// TIA Portal project "ChemicalProcess" (V16)

(* hardware
DEVICE "S71500/ET200MP station_1"  S7-1500 station
   slot 0: "Rail_0"  Rack  6ES7 590-1***0-0AA0
   slot 0: "PS 25W 24VDC_1"  PS 25W 24VDC  6ES7 505-0KA00-0AB0  V1.0
   slot 1: "PLC_1"  CPU 1511-1 PN  6ES7 511-1AK01-0AB0  V2.8
      slot 3: "CPU display_1"  6ES7591-1AA00-0AA0
      slot 32768: "PROFINET interface_1"  X1
         slot 32769: "Port_1"  X1 P1
         slot 32770: "Port_2"  X1 P2
      slot 34817: "Virtual CP interface port_1"  Virtual CP interface port  Virtual CP interface port
   slot 2: "DI 16x24VDC BA_1"  DI 16x24VDC BA  6ES7 521-1BH10-0AA0  V1.1
   slot 3: "DQ 16x24VDC/0.5A BA_1"  DQ 16x24VDC/0.5A BA  6ES7 522-1BH10-0AA0  V1.1
   slot 4: "AI 8xU/I/RTD/TC ST_1"  AI 8xU/I/RTD/TC ST  6ES7 531-7KF00-0AB0  V2.2
   slot 5: "AQ 2xU/I ST_1"  AQ 2xU/I ST  6ES7 532-5NB00-0AB0  V1.0
   slot 6: "DI 16x24VDC BA_2"  DI 16x24VDC BA  6ES7 521-1BH10-0AA0  V1.1
DEVICE "HMI_1"  KTP700 Basic PN
   slot 0: "HMI_1"  KTP700 Basic PN  6AV2 123-2GB03-0AX0  16.0.0.0
   slot 1: "HMI_RT_1"  KTP700 Basic PN  6AV2 123-2GB03-0AX0  16.0.0.0
   slot 5: "HMI_1.IE_CP_1"  PROFINET Interface  16.0.0.0
      slot 1: "PROFINET Interface_1"  PROFINET Interface
         slot 1: "Port_1"  Port
*)

// ===== PLC "PLC_1"  CPU 1511-1 PN =====

VAR_GLOBAL   // PLC tag table "Default tag table"
   "Start" AT %I12.0 : Bool;
   "Stop" AT %I12.1 : Bool;
   "FICSetpoint" AT %MD14 : Real;
END_VAR

VAR_GLOBAL   // PLC tag table "SIMIT interface"
   "ZSO-510" AT %I0.0 : Bool;
   "ZSC-510" AT %I0.1 : Bool;
   "ZSO-511" AT %I0.2 : Bool;
   "ZSC-511" AT %I0.3 : Bool;
   "ZSO-514" AT %I0.4 : Bool;
   "ZSC-514" AT %I0.5 : Bool;
   "ZSO-519" AT %I0.6 : Bool;
   "ZSC-519" AT %I0.7 : Bool;
   "ZSO-521" AT %I1.0 : Bool;
   "ZSC-521" AT %I1.1 : Bool;
   "M001.R" AT %I1.2 : Bool;
   "M002.R" AT %I1.3 : Bool;
   "LS-513" AT %I1.4 : Bool;
   "GSV-510" AT %Q0.0 : Bool;
   "GSV-511" AT %Q0.1 : Bool;
   "GSV-514" AT %Q0.2 : Bool;
   "GSV-519" AT %Q0.3 : Bool;
   "GSV-521" AT %Q0.4 : Bool;
   "M001.ST" AT %Q0.5 : Bool;
   "M002.ST" AT %Q0.6 : Bool;
   "WT-512" AT %IW2 : Int;
   "LT-515" AT %IW4 : Int;
   "FT-516" AT %IW6 : Int;
   "TT-517" AT %IW8 : Int;
   "TT-518" AT %IW10 : Int;
   "M003.SP" AT %QW2 : Int;
   "M001.F" AT %I1.5 : Bool;
   "M002.F" AT %I1.6 : Bool;
   "M003.R" AT %I1.7 : Bool;
   "M003.F" AT %I18.0 : Bool;
   "M003.ST" AT %Q0.7 : Bool;
   "M001.TK" AT %I18.1 : Bool;
   "M002.TK" AT %I18.2 : Bool;
   "M003.TK" AT %I18.3 : Bool;
END_VAR

DATA_BLOCK "ProcessSequence_DB"   // DB3
{ S7_Optimized_Access := 'TRUE' }
VERSION : 0.1
// stored: InstanceOfName ProcessSequence
"ProcessSequence"
BEGIN
END_DATA_BLOCK

DATA_BLOCK "DB_TestMode"   // DB24
{ S7_Optimized_Access := 'TRUE' }
VERSION : 0.1
// stored: InstanceOfName FB_TestMode
"FB_TestMode"
BEGIN
END_DATA_BLOCK

// folder: Motors/Data Blocks

DATA_BLOCK "DB_M001"   // DB10
{ S7_Optimized_Access := 'TRUE' }
VERSION : 0.1
// stored: InstanceOfName FB_Motor
"FB_Motor"
BEGIN
END_DATA_BLOCK

DATA_BLOCK "DB_M002"   // DB14
{ S7_Optimized_Access := 'TRUE' }
VERSION : 0.1
// stored: InstanceOfName FB_Motor
"FB_Motor"
BEGIN
END_DATA_BLOCK

DATA_BLOCK "DB_M003"   // DB18
{ S7_Optimized_Access := 'TRUE' }
VERSION : 0.1
// stored: InstanceOfName FB_Motor
"FB_Motor"
BEGIN
END_DATA_BLOCK

// folder: Process/Data Blocks

DATA_BLOCK "DB_HMI"   // DB19
{ S7_Optimized_Access := 'TRUE' }
VERSION : 0.1
// stored: InstanceOfName FB_HMI
"FB_HMI"
BEGIN
END_DATA_BLOCK

DATA_BLOCK "DB_AutoMode"   // DB20
{ S7_Optimized_Access := 'TRUE' }
VERSION : 0.1
// stored: InstanceOfName FB_Auto
"FB_Auto"
BEGIN
END_DATA_BLOCK

DATA_BLOCK "DB_ManualMode"   // DB21
{ S7_Optimized_Access := 'TRUE' }
VERSION : 0.1
// stored: InstanceOfName FB_Manual
"FB_Manual"
BEGIN
END_DATA_BLOCK

DATA_BLOCK "DB_Stop"   // DB22
{ S7_Optimized_Access := 'TRUE' }
VERSION : 0.1
// stored: InstanceOfName FB_EStop
"FB_EStop"
BEGIN
END_DATA_BLOCK

DATA_BLOCK "DB_Fault"   // DB23
{ S7_Optimized_Access := 'TRUE' }
VERSION : 0.1
// stored: InstanceOfName FB_Fault
"FB_Fault"
BEGIN
END_DATA_BLOCK

// folder: Sensors/DataBlocks

DATA_BLOCK "DB_Sensor_FIC_516"   // DB4
{ S7_Optimized_Access := 'TRUE' }
VERSION : 0.1
// stored: InstanceOfName SensorScaling
"SensorScaling"
BEGIN
END_DATA_BLOCK

DATA_BLOCK "DB_Sensor_WI_512"   // DB12
{ S7_Optimized_Access := 'TRUE' }
VERSION : 0.1
// stored: InstanceOfName SensorScaling
"SensorScaling"
BEGIN
END_DATA_BLOCK

DATA_BLOCK "DB_Sensor_LI_515"   // DB15
{ S7_Optimized_Access := 'TRUE' }
VERSION : 0.1
// stored: InstanceOfName SensorScaling
"SensorScaling"
BEGIN
END_DATA_BLOCK

DATA_BLOCK "Db_Sensor_TI_517"   // DB16
{ S7_Optimized_Access := 'TRUE' }
VERSION : 0.1
// stored: InstanceOfName SensorScaling
"SensorScaling"
BEGIN
END_DATA_BLOCK

DATA_BLOCK "DB_Sensor_TI_518"   // DB17
{ S7_Optimized_Access := 'TRUE' }
VERSION : 0.1
// stored: InstanceOfName SensorScaling
"SensorScaling"
BEGIN
END_DATA_BLOCK

// folder: System blocks/Program resources

DATA_BLOCK "MixTankMotorTImer"   // DB2
{ S7_Optimized_Access := 'TRUE' }
AUTHOR : Simatic
FAMILY : IEC
NAME : IEC_TMR
VERSION : 1.0
// stored: InstanceOfName IEC_TIMER
"IEC_TIMER"
BEGIN
END_DATA_BLOCK

// folder: Valves/DataBlock_Valves

DATA_BLOCK "DB_GSV_510"   // DB5
{ S7_Optimized_Access := 'TRUE' }
VERSION : 0.1
// stored: InstanceOfName FB_Valve
"FB_Valve"
BEGIN
END_DATA_BLOCK

DATA_BLOCK "DB_GSV_511"   // DB6
{ S7_Optimized_Access := 'TRUE' }
VERSION : 0.1
// stored: InstanceOfName FB_Valve
"FB_Valve"
BEGIN
END_DATA_BLOCK

DATA_BLOCK "DB_GSV_514"   // DB7
{ S7_Optimized_Access := 'TRUE' }
VERSION : 0.1
// stored: InstanceOfName FB_Valve
"FB_Valve"
BEGIN
END_DATA_BLOCK

DATA_BLOCK "DB_GSV_519"   // DB8
{ S7_Optimized_Access := 'TRUE' }
VERSION : 0.1
// stored: InstanceOfName FB_Valve
"FB_Valve"
BEGIN
END_DATA_BLOCK

DATA_BLOCK "DB_GSV_521"   // DB9
{ S7_Optimized_Access := 'TRUE' }
VERSION : 0.1
// stored: InstanceOfName FB_Valve
"FB_Valve"
BEGIN
END_DATA_BLOCK

// folder: (top level)

FUNCTION_BLOCK "ProcessSequence"   // FB1, GRAPH_PLUS
{ S7_Optimized_Access := 'TRUE' }
VERSION : 0.1
   VAR_INPUT
      WI_512 : Real;   // WT-512 is Weight Sensor and connected in OB
      LSA_513 : Bool;   // LS-513 Powder Low level Button
      SetTimeForMixing : Time;   // MIx Tank Motor timing
      TI_517 : Real;
      TI_518 : Real;
      FIC_516 : Real;   // FIC-516 is Pressure sensor Integrated with M003
      LI_515 : Real;   // LT-515 Level indicative sensor
      ACK_EF : Bool := false;   // Acknowledge all errors and faults
      Auto : Bool;   // Automode makes sytem run automatically until pressed stop.
      Manual : Bool;   // Manual mode make user start everytime time the storage tank is emptied.
      M003_SP : Real;   // PIDTulo
   END_VAR
   VAR_OUTPUT
      Initiate : Bool;   // Start initiates the program
      HS_510_Open : Bool;   // ZSC-510 is Valve open signal GSV-510.
      HS_510_Close : Bool;   // ZSC-510 Valve close signal for GSV-510.
      GSV_510 : Bool;   // GSV_510 Valve
      HS_511_Open_ : Bool;   // ZSO-511 is Valve open signal GSV-511.
      HS_511_Close : Bool;   // ZSC-511 Valve close signal
      GSV_511 : Bool;   // GSV-511 Valve
      HS_514_Open : Bool;   // ZSO-514 is Valve open signal for GSV-514
      HS_514_Close : Bool;   // ZSC-514 is valve close signal for GSV-514
      GSV_514 : Bool;   // Valve GSV-514.
      HS_519_Open : Bool;   // ZSO-519 is valve open signal for GSV-519
      HS_519_Close : Bool;   // ZSC-519 is Valve close signal for GSV-519
      GSV_519 : Bool;
      HS_521_Open : Bool;   // ZSO-521 valve open signal for GSV-521
      HS_521_Close : Bool;   // ZSC-521 close valve signal for GSV_521
      GSV_521 : Bool;
      SetElapseTimeforMixing : Time;   // Elaspse time for mix tank motor
      M001_ST : Bool;   // M001.ST is Powder Motor start signal.
      M001_TK : Bool;   // M001.TK is Temperature protection of POwder Motor.
      M001_F : Bool;   // M001.F fault signal of Powder Motor
      M001_R : Bool;   // Reset of Powder Motor
      M002_ST : Bool;   // M002.ST is Mixtank Motor signal.
      M002_TK : Bool;
      M002_F : Bool;   // Mator Fault signal For Mix Tank motor
      M002_R : Bool;   // Reset for Mixing Motor
      M003_ST : Bool;   // M003.ST is Start signal of Motor M003
      M003_F : Bool;   // M003.F is Fault signal of Motor M003
      M003_TK : Bool;   // M003.TK isTemperature protection signal of Motor M003
      M003_R : Bool;   // M003.R is Reset signal of Motor M003
      StopandWait : Bool;   // Stop the Process and goest back S and wait until pressed start manually
   END_VAR
   VAR
      HMI_INFO : Array[0..22] of UInt;
      IF_PAR : G7_IfParPlus_V6;
      RT_DATA : G7_RTDataPlus_V6;   // Internal data area
      Trans1 : G7_TransitionPlus_V6;   // Transition structure
      Trans2 : G7_TransitionPlus_V6;   // Transition structure
      Trans3 : G7_TransitionPlus_V6;   // Transition structure
      Trans4 : G7_TransitionPlus_V6;   // Transition structure
      Trans5 : G7_TransitionPlus_V6;   // Transition structure
      Trans6 : G7_TransitionPlus_V6;   // Transition structure
      Trans7 : G7_TransitionPlus_V6;   // Transition structure
      Trans8 : G7_TransitionPlus_V6;   // Transition structure
      Trans9 : G7_TransitionPlus_V6;   // Transition structure
      Trans10 : G7_TransitionPlus_V6;   // Transition structure
      Trans11 : G7_TransitionPlus_V6;   // Transition structure
      Trans12 : G7_TransitionPlus_V6;   // Transition structure
      Start : G7_StepPlus_V6;   // Step structure
      "Fill NaOH" : G7_StepPlus_V6;   // Step structure
      "Fill Powder M001" : G7_StepPlus_V6;   // Step structure
      "Start Mixing" : G7_StepPlus_V6;   // Step structure
      "Empty MIX Tank" : G7_StepPlus_V6;   // Step structure
      "Stop Water" : G7_StepPlus_V6;   // Step structure
      "Close NaOH valve" : G7_StepPlus_V6;   // Step structure
      "Powder Motor Stop" : G7_StepPlus_V6;   // Step structure
      "Stop Mixing" : G7_StepPlus_V6;   // Step structure
      "Empty Storage Tank" : G7_StepPlus_V6;   // Step structure
      "Stop emptying" : G7_StepPlus_V6;   // Step structure
      "Exit valve open" : G7_StepPlus_V6;   // Step structure
      Step13 : G7_StepPlus_V6;   // Step structure
      "Not to Storage" : G7_StepPlus_V6;   // Step structure
      "Exit valve close" : G7_StepPlus_V6;   // Step structure
      "Valve 521 Stays open" : G7_StepPlus_V6;   // Step structure
      "Fill water" : G7_StepPlus_V6;   // Step structure
      Step18 : G7_StepPlus_V6;   // Step structure
      SINI : Array[0..15] of USInt;
      LSTT : Array[0..11] of USInt;
      ATAJ : Array[0..11] of USInt;
      ATAB : Array[0..11] of USInt;
      PSTT : Array[0..11] of USInt;
      NSTT : Array[0..11] of USInt;
      ASSJ : Array[0..17] of USInt;
      ASSB : Array[0..17] of USInt;
      PTTS : Array[0..17] of USInt;
      NTTS : Array[0..17] of USInt;
      SW_SQTS : Array[0..17] of USInt;
      SWITCH : Array[0..36] of USInt;
      TVX : Array[0..15] of USInt;
      TTX : Array[0..15] of USInt;
      TSX : Array[0..15] of USInt;
      S00X : Array[0..15] of USInt;
      SOFFX : Array[0..15] of USInt;
      SONX : Array[0..15] of USInt;
      SAX : Array[0..15] of USInt;
      SERRX : Array[0..18] of USInt;
      SMX : Array[0..18] of USInt;
      S0X : Array[0..18] of USInt;
      S1X : Array[0..18] of USInt;
      IL_ALARM_INST : Diag_Alarm;
      SUP_ALARM_INST : Diag_Alarm;
      STEP_TIME_ALARM_INST : Diag_Alarm;
      IEC_TIMER_INST : IEC_TIMER;
      TRANSACTION_FLAG : Bool := false;
   END_VAR
   // SINI[0] := 2;
   // SINI[2] := 255;
   // SINI[3] := 255;
   // SINI[4] := 255;
   // SINI[5] := 255;
   // SINI[6] := 255;
   // SINI[7] := 255;
   // SINI[8] := 255;
   // SINI[9] := 255;
   // SINI[10] := 255;
   // SINI[11] := 255;
   // SINI[12] := 255;
   // SINI[13] := 255;
   // SINI[14] := 255;
   // SINI[15] := 255;
   // LSTT[0] := 255;
   // LSTT[1] := 255;
   // LSTT[2] := 255;
   // LSTT[3] := 255;
   // LSTT[4] := 255;
   // LSTT[5] := 255;
   // LSTT[7] := 255;
   // LSTT[8] := 255;
   // ATAJ[1] := 1;
   // ATAJ[2] := 2;
   // ATAJ[3] := 3;
   // ATAJ[4] := 4;
   // ATAJ[5] := 5;
   // ATAJ[6] := 6;
   // ATAJ[7] := 7;
   // ATAJ[8] := 8;
   // ATAJ[9] := 9;
   // ATAB[1] := 1;
   // ATAB[2] := 2;
   // ATAB[3] := 3;
   // ATAB[4] := 4;
   // ATAB[5] := 5;
   // ATAB[6] := 6;
   // ATAB[7] := 7;
   // ATAB[8] := 8;
   // ATAB[9] := 9;
   // PSTT[1] := 1;
   // PSTT[2] := 2;
   // PSTT[3] := 3;
   // PSTT[4] := 4;
   // PSTT[5] := 9;
   // PSTT[6] := 10;
   // PSTT[7] := 11;
   // PSTT[8] := 12;
   // PSTT[9] := 14;
   // NSTT[0] := 16;
   // NSTT[1] := 2;
   // NSTT[2] := 3;
   // NSTT[3] := 4;
   // NSTT[4] := 9;
   // NSTT[5] := 11;
   // NSTT[7] := 12;
   // NSTT[8] := 14;
   // ASSJ[1] := 5;
   // ASSJ[2] := 6;
   // ASSJ[3] := 7;
   // ASSJ[4] := 8;
   // ASSJ[5] := 1;
   // ASSJ[6] := 2;
   // ASSJ[7] := 3;
   // ASSJ[8] := 4;
   // ASSJ[9] := 9;
   // ASSJ[10] := 10;
   // ASSJ[11] := 13;
   // ASSJ[12] := 12;
   // ASSJ[13] := 11;
   // ASSJ[14] := 15;
   // ASSJ[15] := 14;
   // ASSB[1] := 5;
   // ASSB[2] := 6;
   // ASSB[3] := 7;
   // ASSB[4] := 8;
   // ASSB[5] := 1;
   // ASSB[6] := 2;
   // ASSB[7] := 3;
   // ASSB[8] := 4;
   // ASSB[9] := 10;
   // ASSB[10] := 9;
   // ASSB[11] := 13;
   // ASSB[12] := 12;
   // ASSB[13] := 11;
   // ASSB[14] := 15;
   // ASSB[15] := 14;
   // PTTS[0] := 255;
   // PTTS[2] := 1;
   // PTTS[3] := 2;
   // PTTS[4] := 3;
   // PTTS[6] := 1;
   // PTTS[7] := 2;
   // PTTS[8] := 3;
   // PTTS[9] := 4;
   // PTTS[10] := 4;
   // PTTS[11] := 5;
   // PTTS[12] := 7;
   // PTTS[13] := 5;
   // PTTS[14] := 8;
   // PTTS[15] := 8;
   // NTTS[1] := 1;
   // NTTS[2] := 2;
   // NTTS[3] := 3;
   // NTTS[4] := 4;
   // NTTS[5] := 1;
   // NTTS[6] := 2;
   // NTTS[7] := 3;
   // NTTS[8] := 4;
   // NTTS[9] := 5;
   // NTTS[10] := 6;
   // NTTS[11] := 7;
   // NTTS[12] := 8;
   // NTTS[13] := 7;
   // NTTS[14] := 9;
   // NTTS[15] := 9;
   // SW_SQTS[1] := 1;
   // SW_SQTS[2] := 2;
   // SW_SQTS[3] := 3;
   // SW_SQTS[4] := 4;
   // SW_SQTS[5] := 5;
   // SW_SQTS[6] := 6;
   // SW_SQTS[7] := 7;
   // SW_SQTS[8] := 8;
   // SW_SQTS[9] := 9;
   // SW_SQTS[10] := 10;
   // SW_SQTS[11] := 11;
   // SW_SQTS[12] := 12;
   // SW_SQTS[13] := 13;
   // SW_SQTS[14] := 14;
   // SW_SQTS[15] := 15;
   // SWITCH[2] := 64;
   // SWITCH[5] := 1;
   // SWITCH[7] := 4;
   // SWITCH[9] := 16;
   // SWITCH[10] := 64;
   // SWITCH[13] := 1;
   // SWITCH[15] := 4;
   // SWITCH[17] := 16;
   // SWITCH[20] := 8;
   // SWITCH[22] := 232;
   // SWITCH[23] := 7;
   // SWITCH[25] := 1;
   // SWITCH[28] := 128;
   // SWITCH[29] := 1;
   // SWITCH[31] := 33;
   // TVX[0] := 16#1;
   // TTX[0] := 16#1;
   // TSX[0] := 16#1;
   // S00X[0] := 16#1;
   // SOFFX[0] := 16#1;
   // SONX[0] := 16#1;
   // SAX[0] := 16#1;
   // SERRX[0] := 16#1;
   // SMX[0] := 16#1;
   // S0X[0] := 16#1;
   // S1X[0] := 16#1;
   // LSTT[10] := 255;
   // ATAJ[10] := 10;
   // ATAB[10] := 10;
   // PSTT[10] := 16;
   // NSTT[10] := 1;
   // ASSJ[16] := 16;
   // ASSB[16] := 16;
   // PTTS[1] := 10;
   // PTTS[5] := 10;
   // NTTS[16] := 10;
   // LSTT[9] := 255;
   // ATAJ[11] := 11;
   // ATAB[11] := 11;
   // PSTT[11] := 17;
   // NSTT[9] := 17;
   // ASSJ[17] := 17;
   // ASSB[17] := 17;
   // PTTS[17] := 9;
   // NTTS[17] := 11;
   // SW_SQTS[17] := 16;
   // SWITCH[24] := 32;
   // SWITCH[26] := 64;
   // SWITCH[33] := 34;
   // SWITCH[35] := 4;
BEGIN
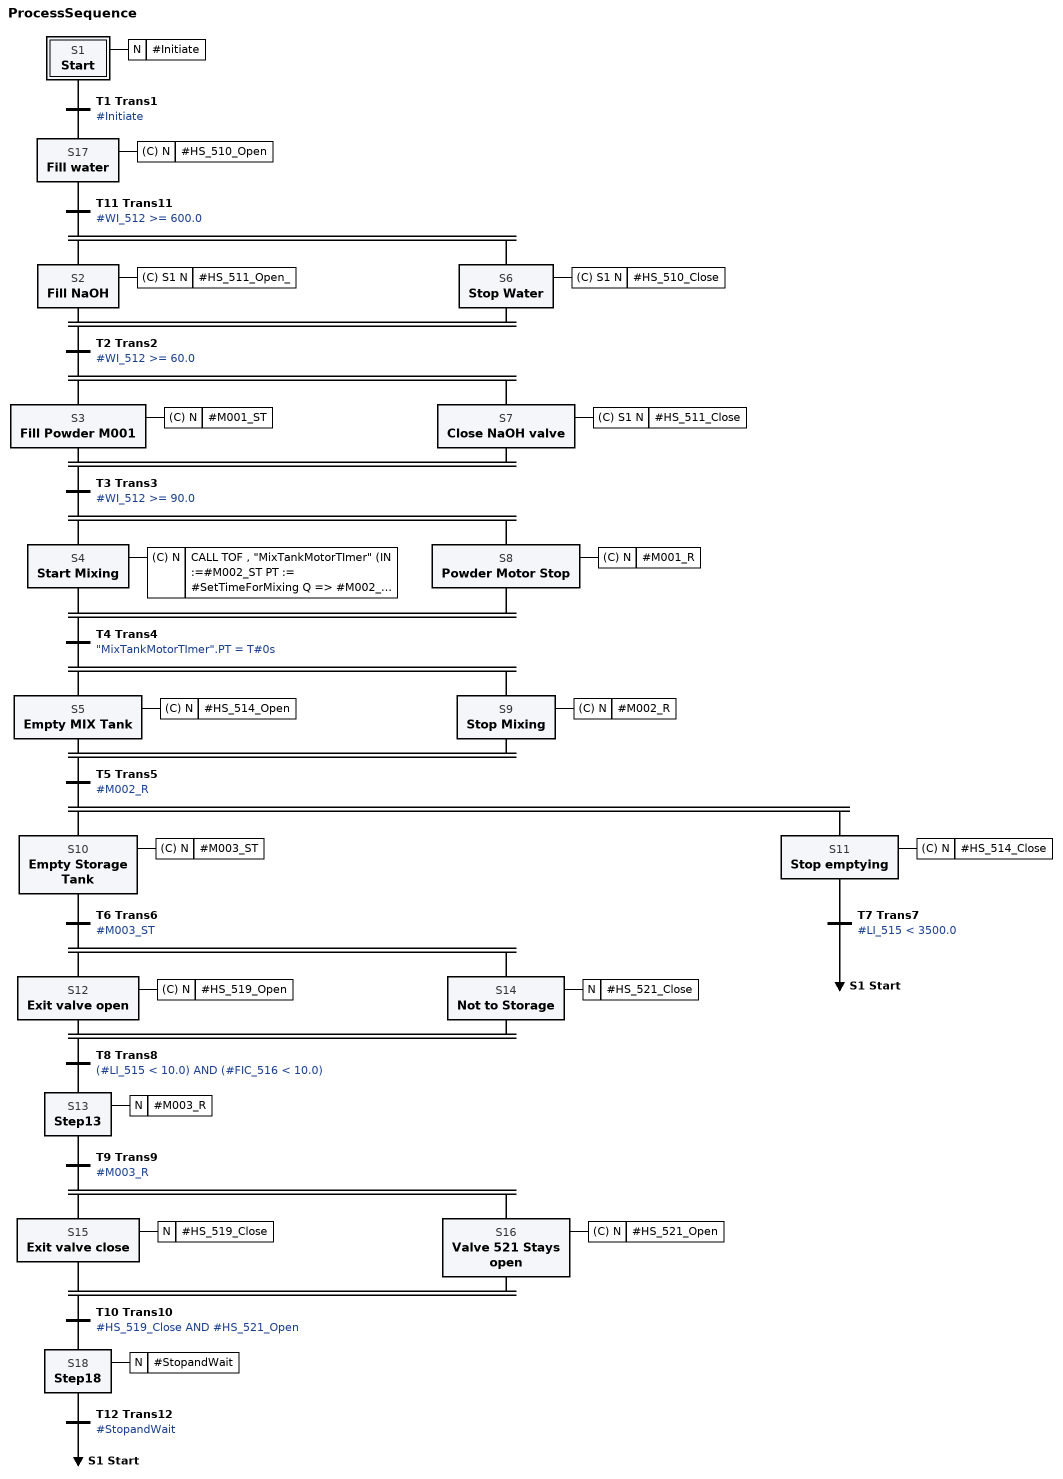
   // sequencer 1
   INITIAL_STEP Start:   // S1, max time T#10S, warning time T#7S
      interlock C := ((#Auto AND NOT #Manual) OR (#Manual AND NOT #Auto)) AND NOT #StopandWait;
              N    #Initiate
   END_STEP
   TRANSITION Trans1 FROM Start TO "Fill water"   // T1
      := #Initiate;
   END_TRANSITION
   STEP "Fill NaOH":   // S2, max time T#10S, warning time T#7S
      interlock C := (#WI_512 <= 40.0) AND NOT #GSV_510 AND NOT #M001_ST AND NOT #M002_ST;
      // 600Kg to 1200kg in weight sensor is 600Kg of NaOH.
      (C) S1  N    #HS_511_Open_
   END_STEP
   STEP "Fill Powder M001":   // S3, max time T#10S, warning time T#7S
      interlock C := NOT #GSV_510 AND NOT #M002_ST AND NOT #LSA_513 AND NOT #M001_F AND NOT #M001_TK AND NOT #GSV_511;
      // 1200-1800KG in wight sensor = 600Kg of Powder
      (C)     N    #M001_ST
   END_STEP
   STEP "Start Mixing":   // S4, max time T#10S, warning time T#7S
      interlock C := NOT #GSV_510 AND NOT #GSV_511 AND NOT #M001_ST AND NOT #M002_F;
      (C)     N    CALL TOF , "MixTankMotorTImer"
                   (IN :=#M002_ST
                   PT := #SetTimeForMixing
                   Q => #M002_R
                   ET=> #SetElapseTimeforMixing
                   )
   END_STEP
   STEP "Empty MIX Tank":   // S5, max time T#10S, warning time T#7S
      interlock C := (#LI_515 < 80.0) AND NOT #GSV_510 AND NOT #GSV_511 AND NOT #M002_ST AND NOT #M001_ST;
      (C)     N    #HS_514_Open
   END_STEP
   STEP "Stop Water":   // S6, max time T#10S, warning time T#7S
      interlock C := #WI_512 >= 30.0;
      // If Valve opens have to make sure it closes.
      (C) S1  N    #HS_510_Close
   END_STEP
   TRANSITION Trans2 FROM ("Fill NaOH", "Stop Water") TO ("Fill Powder M001", "Close NaOH valve")   // T2
      := #WI_512 >= 60.0;
   END_TRANSITION
   STEP "Close NaOH valve":   // S7, max time T#10S, warning time T#7S
      interlock C := #WI_512 = 60.0;
      (C) S1  N    #HS_511_Close
   END_STEP
   TRANSITION Trans3 FROM ("Fill Powder M001", "Close NaOH valve") TO ("Start Mixing", "Powder Motor Stop")   // T3
      := #WI_512 >= 90.0;
   END_TRANSITION
   STEP "Powder Motor Stop":   // S8, max time T#10S, warning time T#7S
      interlock C := #WI_512 >= 90.0;
      (C)     N    #M001_R
   END_STEP
   TRANSITION Trans4 FROM ("Start Mixing", "Powder Motor Stop") TO ("Empty MIX Tank", "Stop Mixing")   // T4
      := "MixTankMotorTImer".PT = T#0s;
   END_TRANSITION
   STEP "Stop Mixing":   // S9, max time T#10S, warning time T#7S
      interlock C := "MixTankMotorTImer".PT = T#0s;
      (C)     N    #M002_R
   END_STEP
   TRANSITION Trans5 FROM ("Empty MIX Tank", "Stop Mixing") TO ("Empty Storage Tank", "Stop emptying")   // T5
      := #M002_R;
   END_TRANSITION
   STEP "Empty Storage Tank":   // S10, max time T#10S, warning time T#7S
      interlock C := NOT #GSV_514 AND (#LI_515 > 70.0) AND NOT #M003_F AND NOT #M003_TK AND NOT #M003_R;
      (C)     N    #M003_ST
   END_STEP
   TRANSITION Trans6 FROM "Empty Storage Tank" TO ("Exit valve open", "Not to Storage")   // T6
      := #M003_ST;
   END_TRANSITION
   STEP "Stop emptying":   // S11, max time T#10S, warning time T#7S
      interlock C := #WI_512 <= 2.0;   // Stop Emptying
      (C)     N    #HS_514_Close
   END_STEP
   TRANSITION Trans7 FROM "Stop emptying" TO Start   // T7, jump
      := #LI_515 < 3500.0;
   END_TRANSITION
   STEP "Exit valve open":   // S12, max time T#10S, warning time T#7S
      interlock C := #M003_ST;
      (C)     N    #HS_519_Open
   END_STEP
   STEP Step13:   // S13, max time T#10S, warning time T#7S
      interlock C := (#LI_515 < 5.0) AND (#FIC_516 < 5.0);
              N    #M003_R
   END_STEP
   TRANSITION Trans9 FROM Step13 TO ("Exit valve close", "Valve 521 Stays open")   // T9
      := #M003_R;
   END_TRANSITION
   STEP "Not to Storage":   // S14, max time T#10S, warning time T#7S
      interlock C := #M003_ST;
              N    #HS_521_Close
   END_STEP
   TRANSITION Trans8 FROM ("Exit valve open", "Not to Storage") TO Step13   // T8
      := (#LI_515 < 10.0) AND (#FIC_516 < 10.0);
   END_TRANSITION
   STEP "Exit valve close":   // S15, max time T#10S, warning time T#7S
      interlock C := #M003_R AND (#FIC_516 < 5.0);
              N    #HS_519_Close
   END_STEP
   STEP "Valve 521 Stays open":   // S16, max time T#10S, warning time T#7S
      interlock C := #M003_R AND (#FIC_516 < 5.0);
      (C)     N    #HS_521_Open
   END_STEP
   TRANSITION Trans10 FROM ("Exit valve close", "Valve 521 Stays open") TO Step18   // T10
      := #HS_519_Close AND #HS_521_Open;
   END_TRANSITION
   STEP "Fill water":   // S17, max time T#10S, warning time T#7S
      interlock C := (#WI_512 <= 5.0) AND NOT #HS_510_Close AND NOT #GSV_511 AND NOT #M001_ST AND NOT #M002_ST;
      // 1Litre = 1Kg, 0-600Kg in Weight sensor is 600litres of Water For forcing value of sensors converts kg value to Siemens analog raw value (0...27648). For 200KG = 2765
      (C)     N    #HS_510_Open
   END_STEP
   TRANSITION Trans11 FROM "Fill water" TO ("Fill NaOH", "Stop Water")   // T11
      := #WI_512 >= 600.0;
   END_TRANSITION
   STEP Step18:   // S18, max time T#10S, warning time T#7S
              N    #StopandWait
   END_STEP
   TRANSITION Trans12 FROM Step18 TO Start   // T12, jump
      := #StopandWait;
   END_TRANSITION
END_FUNCTION_BLOCK

FUNCTION_BLOCK "FB_TestMode"   // FB9, FBD
{ S7_Optimized_Access := 'TRUE' }
VERSION : 0.1
   VAR_INPUT
      TestOn : Bool;   // Test mode enable
      TestOff : Bool;
   END_VAR
   VAR_OUTPUT
      Valve1 : Bool;
      Valve2 : Bool;
      Valve3 : Bool;
      Valve4 : Bool;
      Valve5 : Bool;
      Motor1 : Bool;
      Motor2 : Bool;
      Motor3 : Bool;
   END_VAR
   VAR
      TestRSmemory : Bool;
   END_VAR
BEGIN

REGION Network 1
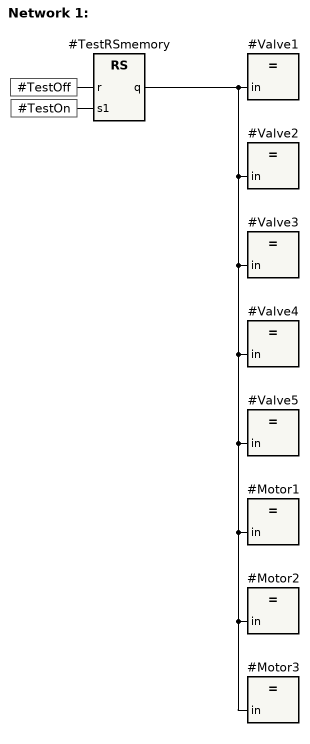
   IF #TestOff THEN
       #TestRSmemory := FALSE;   // RS flip-flop
   END_IF;
   IF #TestOn THEN #TestRSmemory := TRUE; END_IF;
   #Valve1 := #TestRSmemory;
   #Valve2 := #TestRSmemory;
   #Valve3 := #TestRSmemory;
   #Valve4 := #TestRSmemory;
   #Valve5 := #TestRSmemory;
   #Motor1 := #TestRSmemory;
   #Motor2 := #TestRSmemory;
   #Motor3 := #TestRSmemory;
END_REGION
END_FUNCTION_BLOCK

ORGANIZATION_BLOCK "Main"   // OB1, FBD, ProgramCycle
TITLE = "Main Program Sweep (Cycle)"
{ S7_Optimized_Access := 'TRUE' }
VERSION : 0.1
// This is where physical world meets the digital world.
// Main cyclic control block. Calls HMI handling, operating modes, safety/fault logic, sensor scaling, actuator control, and process sequence in defined order.
   VAR_INPUT
      Initial_Call : Bool;   // Initial call of this OB
      Remanence : Bool;   // =True, if remanent data are available
   END_VAR
   VAR_TEMP
      Scaled_WI512 : Real;   // WT/WI-512 sensor´s scaled value.
      Scaled_LI515 : Real;   // LT/LI-515 sensor´s scaled value
      Scaled_TI517 : Real;   // TT/TI-517 sensor´s scaled value
      Scaled_TI518 : Real;   // TT/TI-518 sensor´s scaled value
      Scaled_FIC516 : Real;   // Current sensor for PumpM003
      M003ScaledStatus : Word;
   END_VAR
BEGIN

REGION Network 1: HMI
   // Not in use for now. Reads operator commands and prepares start, stop, reset, auto/manual selections.
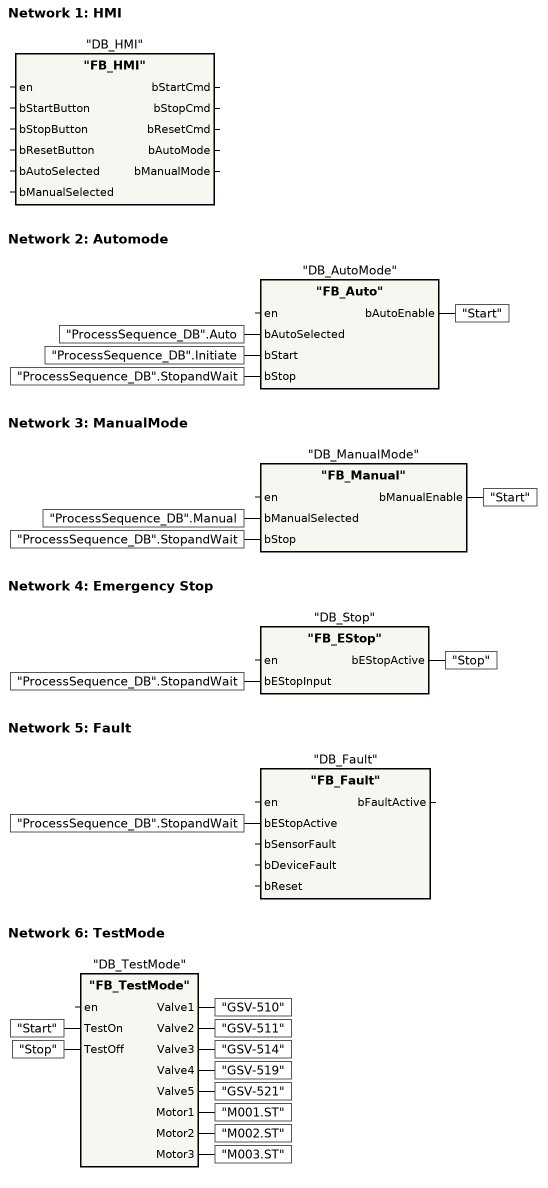
   "DB_HMI"();   // "FB_HMI"
END_REGION

REGION Network 2: Automode
   // Creates automatic operation enable signal from HMI mode selection and start/stop commands.
   "DB_AutoMode"(bAutoSelected := "ProcessSequence_DB".Auto,   // "FB_Auto"
                 bStart := "ProcessSequence_DB".Initiate,
                 bStop := "ProcessSequence_DB".StopandWait,
                 bAutoEnable => "Start");
END_REGION

REGION Network 3: ManualMode
   // Creates manual operation enable signal for direct operator-controlled device operation.
   "DB_ManualMode"(bManualSelected := "ProcessSequence_DB".Manual,   // "FB_Manual"
                   bStop := "ProcessSequence_DB".StopandWait,
                   bManualEnable => "Start");
END_REGION

REGION Network 4: Emergency Stop
   // Processes emergency stop input and creates global emergency stop active signal.
   "DB_Stop"(bEStopInput := "ProcessSequence_DB".StopandWait, bEStopActive => "Stop");   // "FB_EStop"
END_REGION

REGION Network 5: Fault
   // Collects process, device, sensor, and emergency stop faults into one fault status.
   "DB_Fault"(bEStopActive := "ProcessSequence_DB".StopandWait);   // "FB_Fault"
END_REGION

REGION Network 6: TestMode
   // Creates global all outputs ON/OFF test commands.
   "DB_TestMode"(TestOn := "Start",   // "FB_TestMode"
                 TestOff := "Stop",
                 Valve1 => "GSV-510",
                 Valve2 => "GSV-511",
                 Valve3 => "GSV-514",
                 Valve4 => "GSV-519",
                 Valve5 => "GSV-521",
                 Motor1 => "M001.ST",
                 Motor2 => "M002.ST",
                 Motor3 => "M003.ST");
END_REGION

REGION Network 7: Sensors Scalings
   // Scales raw analog sensor values into engineering units for process logic.
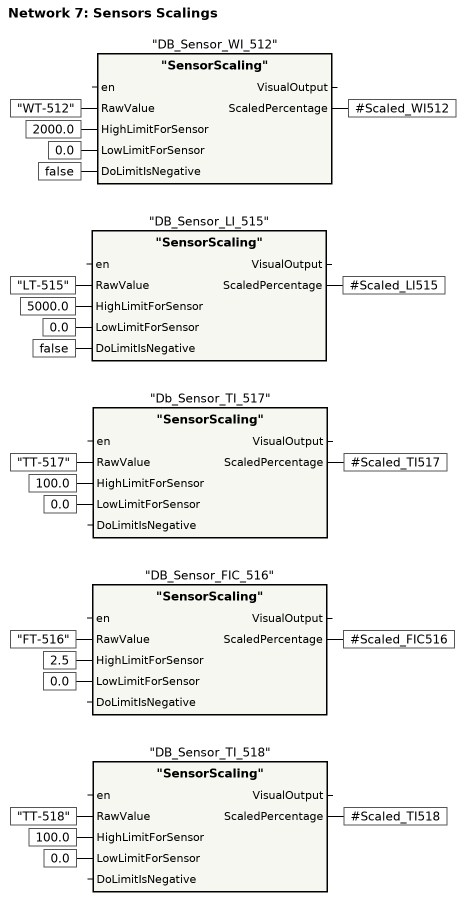
   "DB_Sensor_WI_512"(RawValue := "WT-512",   // "SensorScaling"
                      HighLimitForSensor := 2000.0,
                      LowLimitForSensor := 0.0,
                      DoLimitIsNegative := false,
                      ScaledPercentage => #Scaled_WI512);
   "DB_Sensor_LI_515"(RawValue := "LT-515",   // "SensorScaling"
                      HighLimitForSensor := 5000.0,
                      LowLimitForSensor := 0.0,
                      DoLimitIsNegative := false,
                      ScaledPercentage => #Scaled_LI515);
   "Db_Sensor_TI_517"(RawValue := "TT-517",   // "SensorScaling"
                      HighLimitForSensor := 100.0,
                      LowLimitForSensor := 0.0,
                      ScaledPercentage => #Scaled_TI517);
   "DB_Sensor_FIC_516"(RawValue := "FT-516",   // "SensorScaling"
                       HighLimitForSensor := 2.5,
                       LowLimitForSensor := 0.0,
                       ScaledPercentage => #Scaled_FIC516);
   "DB_Sensor_TI_518"(RawValue := "TT-518",   // "SensorScaling"
                      HighLimitForSensor := 100.0,
                      LowLimitForSensor := 0.0,
                      ScaledPercentage => #Scaled_TI518);
END_REGION

REGION Network 8: PID FIC-516 /M003
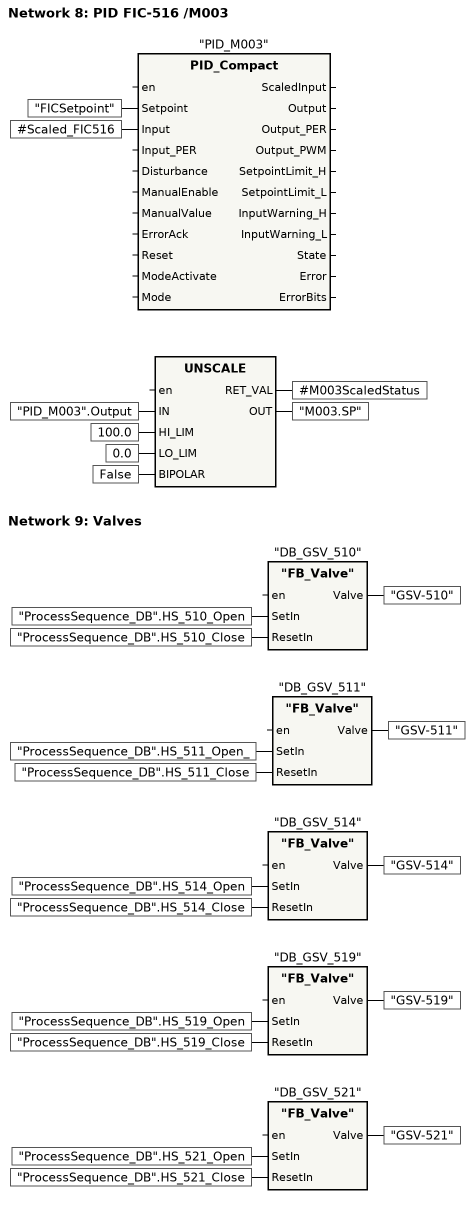
   "PID_M003"(Setpoint := "FICSetpoint", Input := #Scaled_FIC516);   // PID_Compact
   #M003ScaledStatus := UNSCALE(IN := "PID_M003".Output,
                           HI_LIM := 100.0,
                           LO_LIM := 0.0,
                           BIPOLAR := False,
                           OUT => "M003.SP");
END_REGION

REGION Network 9: Valves
   // Calls valve FB instances and maps sequence/manual commands to physical valve outputs.
   "DB_GSV_510"(SetIn := "ProcessSequence_DB".HS_510_Open,   // "FB_Valve"
                ResetIn := "ProcessSequence_DB".HS_510_Close,
                Valve => "GSV-510");
   "DB_GSV_511"(SetIn := "ProcessSequence_DB".HS_511_Open_,   // "FB_Valve"
                ResetIn := "ProcessSequence_DB".HS_511_Close,
                Valve => "GSV-511");
   "DB_GSV_514"(SetIn := "ProcessSequence_DB".HS_514_Open,   // "FB_Valve"
                ResetIn := "ProcessSequence_DB".HS_514_Close,
                Valve => "GSV-514");
   "DB_GSV_519"(SetIn := "ProcessSequence_DB".HS_519_Open,   // "FB_Valve"
                ResetIn := "ProcessSequence_DB".HS_519_Close,
                Valve => "GSV-519");
   "DB_GSV_521"(SetIn := "ProcessSequence_DB".HS_521_Open,   // "FB_Valve"
                ResetIn := "ProcessSequence_DB".HS_521_Close,
                Valve => "GSV-521");
END_REGION

REGION Network 10: Motors
   // Calls motor FB instances and maps sequence/manual commands to physical motor outputs.
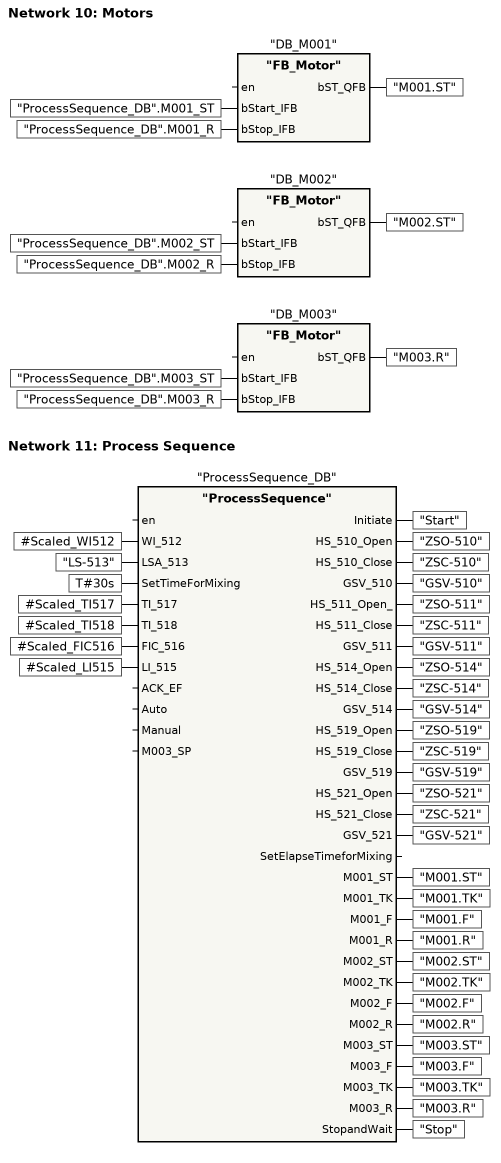
   "DB_M001"(bStart_IFB := "ProcessSequence_DB".M001_ST,   // "FB_Motor"
             bStop_IFB := "ProcessSequence_DB".M001_R,
             bST_QFB => "M001.ST");
   "DB_M002"(bStart_IFB := "ProcessSequence_DB".M002_ST,   // "FB_Motor"
             bStop_IFB := "ProcessSequence_DB".M002_R,
             bST_QFB => "M002.ST");
   "DB_M003"(bStart_IFB := "ProcessSequence_DB".M003_ST,   // "FB_Motor"
             bStop_IFB := "ProcessSequence_DB".M003_R,
             bST_QFB => "M003.R");
END_REGION

REGION Network 11: Process Sequence
   // Runs GRAPH process sequence for automatic batch operation.
   "ProcessSequence_DB"(WI_512 := #Scaled_WI512,   // "ProcessSequence"
                        LSA_513 := "LS-513",
                        SetTimeForMixing := T#30s,
                        TI_517 := #Scaled_TI517,
                        TI_518 := #Scaled_TI518,
                        FIC_516 := #Scaled_FIC516,
                        LI_515 := #Scaled_LI515,
                        Initiate => "Start",
                        HS_510_Open => "ZSO-510",
                        HS_510_Close => "ZSC-510",
                        GSV_510 => "GSV-510",
                        HS_511_Open_ => "ZSO-511",
                        HS_511_Close => "ZSC-511",
                        GSV_511 => "GSV-511",
                        HS_514_Open => "ZSO-514",
                        HS_514_Close => "ZSC-514",
                        GSV_514 => "GSV-514",
                        HS_519_Open => "ZSO-519",
                        HS_519_Close => "ZSC-519",
                        GSV_519 => "GSV-519",
                        HS_521_Open => "ZSO-521",
                        HS_521_Close => "ZSC-521",
                        GSV_521 => "GSV-521",
                        M001_ST => "M001.ST",
                        M001_TK => "M001.TK",
                        M001_F => "M001.F",
                        M001_R => "M001.R",
                        M002_ST => "M002.ST",
                        M002_TK => "M002.TK",
                        M002_F => "M002.F",
                        M002_R => "M002.R",
                        M003_ST => "M003.ST",
                        M003_F => "M003.F",
                        M003_TK => "M003.TK",
                        M003_R => "M003.R",
                        StopandWait => "Stop");
END_REGION

REGION Network 12: Spare/Future Expansion
   // Reserved for future PID, VFD, alarms, diagnostics, or reporting logic.
END_REGION
END_ORGANIZATION_BLOCK

// folder: Motors/Generic Motors

FUNCTION_BLOCK "FB_Motor"   // FB11, FBD
{ S7_Optimized_Access := 'TRUE' }
VERSION : 0.1
   VAR_INPUT
      bStart_IFB : Bool;
      bStop_IFB : Bool;
   END_VAR
   VAR_OUTPUT
      bST_QFB : Bool;
   END_VAR
   VAR_TEMP
      Reset : Bool;
      Set : Bool;
   END_VAR
BEGIN

REGION Network 1
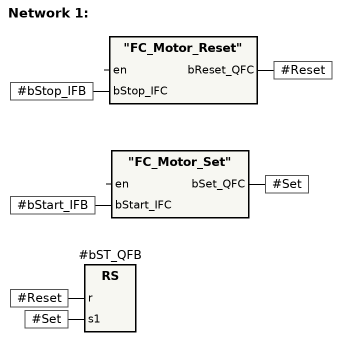
   "FC_Motor_Reset"(bStop_IFC := #bStop_IFB, bReset_QFC => #Reset);
   "FC_Motor_Set"(bStart_IFC := #bStart_IFB, bSet_QFC => #Set);
   IF #Reset THEN
       #bST_QFB := FALSE;   // RS flip-flop
   END_IF;
   IF #Set THEN #bST_QFB := TRUE; END_IF;
END_REGION
END_FUNCTION_BLOCK

FUNCTION "FC_Motor_Set" : Void   // FC5, FBD
{ S7_Optimized_Access := 'TRUE' }
VERSION : 0.1
   VAR_INPUT
      bStart_IFC : Bool;   // Start request for motor
   END_VAR
   VAR_OUTPUT
      bSet_QFC : Bool;   // Set signal to motor memory
   END_VAR
BEGIN

REGION Network 1: Set signal to motor memory
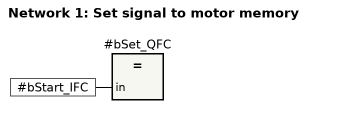
   #bSet_QFC := #bStart_IFC;
END_REGION
END_FUNCTION

FUNCTION "FC_Motor_Reset" : Void   // FC6, FBD
{ S7_Optimized_Access := 'TRUE' }
VERSION : 0.1
   VAR_INPUT
      bStop_IFC : Bool;   // Stop request for motor
   END_VAR
   VAR_OUTPUT
      bReset_QFC : Bool;   // Reset signal to motor memory
   END_VAR
BEGIN

REGION Network 1: Reset output
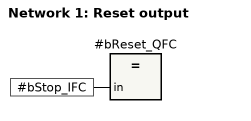
   #bReset_QFC := #bStop_IFC;
END_REGION
END_FUNCTION

// folder: Process/Process FBs

FUNCTION_BLOCK "FB_Auto"   // FB4, FBD
{ S7_Optimized_Access := 'TRUE' }
VERSION : 0.1
   VAR_INPUT
      bAutoSelected : Bool;
      bStart : Bool;
      bStop : Bool;
   END_VAR
   VAR_OUTPUT
      bAutoEnable : Bool;
   END_VAR
BEGIN

REGION Network 1
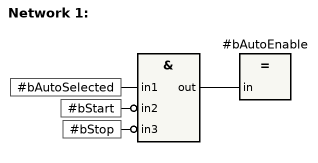
   #bAutoEnable := #bAutoSelected AND NOT #bStart AND NOT #bStop;
END_REGION
END_FUNCTION_BLOCK

FUNCTION_BLOCK "FB_Manual"   // FB5, FBD
{ S7_Optimized_Access := 'TRUE' }
VERSION : 0.1
   VAR_INPUT
      bManualSelected : Bool;
      bStop : Bool;
   END_VAR
   VAR_OUTPUT
      bManualEnable : Bool;
   END_VAR
BEGIN

REGION Network 1
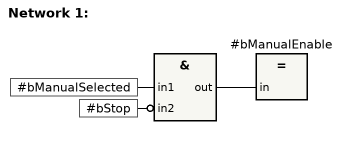
   #bManualEnable := #bManualSelected AND NOT #bStop;
END_REGION
END_FUNCTION_BLOCK

FUNCTION_BLOCK "FB_EStop"   // FB6, FBD
{ S7_Optimized_Access := 'TRUE' }
VERSION : 0.1
   VAR_INPUT
      bEStopInput : Bool;
   END_VAR
   VAR_OUTPUT
      bEStopActive : Bool;
   END_VAR
BEGIN

REGION Network 1
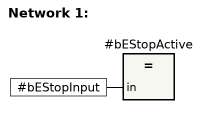
   #bEStopActive := #bEStopInput;
END_REGION
END_FUNCTION_BLOCK

FUNCTION_BLOCK "FB_Fault"   // FB7, FBD
{ S7_Optimized_Access := 'TRUE' }
VERSION : 0.1
   VAR_INPUT
      bEStopActive : Bool;
      bSensorFault : Bool;
      bDeviceFault : Bool;
      bReset : Bool;
   END_VAR
   VAR_OUTPUT
      bFaultActive : Bool;
   END_VAR
BEGIN

REGION Network 1
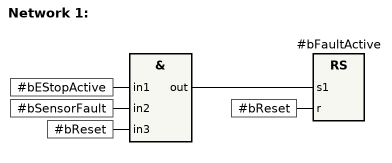
   IF #bReset THEN
       #bFaultActive := FALSE;   // RS flip-flop
   END_IF;
   IF #bEStopActive AND #bSensorFault AND #bReset THEN #bFaultActive := TRUE; END_IF;
END_REGION
END_FUNCTION_BLOCK

FUNCTION_BLOCK "FB_HMI"   // FB8, FBD
{ S7_Optimized_Access := 'TRUE' }
VERSION : 0.1
   VAR_INPUT
      bStartButton : Bool;
      bStopButton : Bool;
      bResetButton : Bool;
      bAutoSelected : Bool;
      bManualSelected : Bool;
   END_VAR
   VAR_OUTPUT
      bStartCmd : Bool;
      bStopCmd : Bool;
      bResetCmd : Bool;
      bAutoMode : Bool;
      bManualMode : Bool;
   END_VAR
BEGIN
END_FUNCTION_BLOCK

// folder: Sensors/Generic Blocks

FUNCTION_BLOCK "SensorScaling"   // FB3, FBD
TITLE = Sensor Fb Block
{ S7_Optimized_Access := 'TRUE' }
VERSION : 0.1
// The idea is to call this from FC and then call it into OB and connect sensors individually, by doing that DB instance can be created for sensors and  everythin will be connected inside one and highest layer, this will help in maintenance, monitoring, optimization, further analysis and future possiblities.
   VAR_INPUT
      RawValue : Int;   // Connect the sensor Straight here. 4-20mA = 0-27648 Integers.
      HighLimitForSensor : Real;   // High limit required in plan
      LowLimitForSensor : Real;   // Low limit required in plan
      DoLimitIsNegative : Bool;   // If limit is negative then Bipolar:= true elseif positive then unipolar:= true
   END_VAR
   VAR_OUTPUT
      VisualOutput : Word;   // Visual Output for further use.
      ScaledPercentage : Real;
   END_VAR
   VAR
      Result : Real;
      ActualOutput : Real;   // Usable output for futher use.
   END_VAR
BEGIN

REGION Network 1
   // Basic FC to FB call.
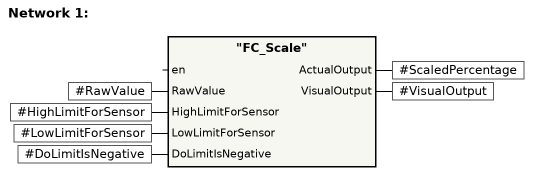
   "FC_Scale"(RawValue := #RawValue,
              HighLimitForSensor := #HighLimitForSensor,
              LowLimitForSensor := #LowLimitForSensor,
              DoLimitIsNegative := #DoLimitIsNegative,
              ActualOutput => #ScaledPercentage,
              VisualOutput => #VisualOutput);
END_REGION
END_FUNCTION_BLOCK

FUNCTION "FC_Scale" : Void   // FC2, FBD
TITLE = Scaling for Sensors
{ S7_Optimized_Access := 'TRUE' }
VERSION : 0.1
// This is a basic mechanism for scaling Sensors. For details about using Function scale, visit this website https://support.industry.siemens.com/cs/document/1765297/how-and-for-which-analog-measurements-can-you-use-the-function-fc105-scale-to-convert-the-integer-values-(int)-into-real-number-values-?dti=0&lc=en-SZ
   VAR_INPUT
      RawValue : Int;   // Connect the sensor Straight here. 4-20mA = 0-27648 Integers.
      HighLimitForSensor : Real;   // High limit required in plan
      LowLimitForSensor : Real;   // Low limit required in plan
      DoLimitIsNegative : Bool;   // If limit is negative then Bipolar:= true elseif positive then unipolar:= true
   END_VAR
   VAR_OUTPUT
      ActualOutput : Real;   // Usable output for futher use.
      VisualOutput : Word;   // Visual Output for further use.
   END_VAR
BEGIN

REGION Network 1
   // Basci scale block
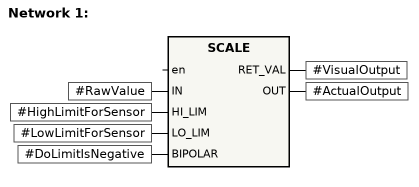
   #VisualOutput := SCALE(IN := #RawValue,
                          HI_LIM := #HighLimitForSensor,
                          LO_LIM := #LowLimitForSensor,
                          BIPOLAR := #DoLimitIsNegative,
                          OUT => #ActualOutput);
END_REGION
END_FUNCTION

// folder: Valves/Generic valves

FUNCTION_BLOCK "FB_Valve"   // FB2, FBD
{ S7_Optimized_Access := 'TRUE' }
VERSION : 0.1
   VAR_INPUT
      SetIn : Bool;
      ResetIn : Bool;
   END_VAR
   VAR_OUTPUT
      Valve : Bool;
   END_VAR
   VAR_TEMP
      SetOutput : Bool;
      ResetOutput : Bool;
   END_VAR
BEGIN

REGION Network 1
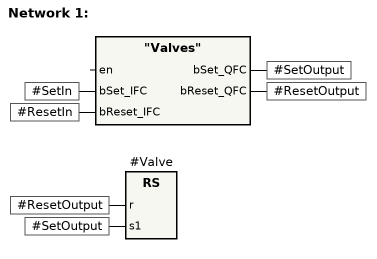
   "Valves"(bSet_IFC := #SetIn, bReset_IFC := #ResetIn, bSet_QFC => #SetOutput, bReset_QFC => #ResetOutput);
   IF #ResetOutput THEN
       #Valve := FALSE;   // RS flip-flop
   END_IF;
   IF #SetOutput THEN #Valve := TRUE; END_IF;
END_REGION
END_FUNCTION_BLOCK

FUNCTION "Valves" : Void   // FC1, FBD
{ S7_Optimized_Access := 'TRUE' }
VERSION : 0.1
   VAR_INPUT
      bSet_IFC : Bool;   // Set valve open command
      bReset_IFC : Bool;   // Reset valve close command
   END_VAR
   VAR_OUTPUT
      bSet_QFC : Bool;   // Set signal to valve memory
      bReset_QFC : Bool;   // Reset signal to valve memory
   END_VAR
BEGIN

REGION Network 1: Set signal to valve memory
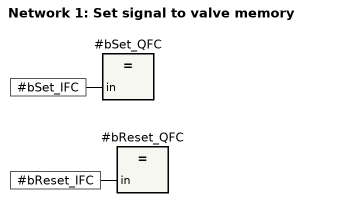
   #bSet_QFC := #bSet_IFC;
   #bReset_QFC := #bReset_IFC;
END_REGION
END_FUNCTION

(* ===== HMI "HMI_RT_1" =====
system functions are stored by id; their names below are inferred from use
connection "HMI_Connection_1": ETHERNET, SMART_S7_1500_OMS

HMI tags "Default tag table"
   "Tag_ScreenNumber" : UInt, internal
   "WT-512" : Int = PLC "WT-512" AT %IW2, 1 s
   "GSV-510" : Bool = PLC "GSV-510" AT %Q0.0, 1 s
   "GSV-511" : Bool = PLC "GSV-511" AT %Q0.1, 1 s
   "GSV-514" : Bool = PLC "GSV-514" AT %Q0.2, 1 s
   "GSV-519" : Bool = PLC "GSV-519" AT %Q0.3, 1 s
   "GSV-521" : Bool = PLC "GSV-521" AT %Q0.4, 1 s
   "M001.ST" : Bool = PLC "M001.ST" AT %Q0.5, 1 s
   "M002.ST" : Bool = PLC "M002.ST" AT %Q0.6, 1 s
   "M003.ST" : Bool = PLC "M003.ST" AT %Q0.7, 1 s
   "TT-518" : Int = PLC "TT-518" AT %IW10, 1 s
   "TT-517" : Int = PLC "TT-517" AT %IW8, 1 s
   "LT-515" : Int = PLC "LT-515" AT %IW4, 1 s
   "LS-513" : Bool = PLC "LS-513" AT %I1.4, 1 s
   "M001.R" : Bool = PLC "M001.R" AT %I1.2, 1 s
   "M002.R" : Bool = PLC "M002.R" AT %I1.3, 1 s
   "M003.R" : Bool = PLC "M003.R" AT %I1.7, 1 s

Template "Template_1" 800x480
   Button "Exit" at 714,429 size 71x50; TextOff 'Exit'; PictureOff "ExitRuntime_KTP700_Basic_PN_TR"; PictureOn "ExitRuntime_KTP700_Basic_PN_TR"
      on Release: StopRuntime(0)
   Button "Language" at 614,429 size 71x50; TextOff 'Language'; PictureOff "ToggleLanguage_KTP700_Basic_PN_TR"; PictureOn "ToggleLanguage_KTP700_Basic_PN_TR"
      on Release: function_fb9197e8(-1)
   Button "Template_Button" at 514,429 size 71x50; TextOff 'Text'
   Button "Template_Button_1" at 414,429 size 71x50; TextOff 'Text'
   Button "Template_Button_2" at 314,429 size 71x50; TextOff 'Text'
   Button "Template_Button_3" at 214,429 size 71x50; TextOff 'Text'
   Button "Alarms" at 114,429 size 71x50; TextOff 'Alarms'; PictureOff "AlarmDisplay_KTP700_Basic_PN_TR"; PictureOn "AlarmDisplay_KTP700_Basic_PN_TR"
      on Release: function_ef3f5d25("Alarm window_Unacknowledged", -1)
   Button "Start screen" at 14,429 size 71x50; TextOff 'Start screen'; PictureOff "NavigateHome_KTP700_Basic_PN_TR"; PictureOn "NavigateHome_KTP700_Basic_PN_TR"
      on Release: ActivateScreen("Root screen", 0)
   SymbolicIOField "Symbolic_IO_Field_Screen" at 93,9 size 600x33; TextOff '0'; TextOn '1'; TextList "TextList_ScreenNames"
      ProcessValue <- "Tag_ScreenNumber"
      on Change: ActivateScreenByNumber("Tag_ScreenNumber", 0)
   DateTimeField "HmiScreenItemData" at 695,25 size 105x25
   DateTimeField "HmiScreenItemData_1" at 695,0 size 105x25
   GraphicView "Logo" at 0,0 size 91x51; Picture "Logo of HMI_1"

screen "Root screen" 800x480, template "Template_1"
   on GenerateScreen: SetTag("Tag_ScreenNumber", 1)
   Button "HmiScreenItemData_1" at 623,67 size 159x47; TextOff 'System screens'; PictureOff "Navigates to System screens for KTP700 Basic+ PN 16.0.0.0"; PictureOn "Navigates to System screens for KTP700 Basic+ PN 16.0.0.0"
      on Release: ActivateScreen("System screens", 0)
   IOField "I/O field_1" at 120,129 size 96x32; FormatPattern s999
      ProcessValue <- "WT-512"
   TextField "Text field_1" at 42,137 size 65x23; Text 'WI-512'
   Switch "Switch_1" at 357,120 size 64x32; CaptionText 'Switch'; TextOff 'OFF'; TextOn 'ON'
      ProcessValue <- "GSV-510"
   TextField "Text field_3" at 283,122 size 16x23; Text 'Text'
   TextField "Text field_2" at 277,122 size 75x23; Text 'GSV-510'
   Switch "Switch_2" at 357,168 size 64x32; TextOn 'ON'; CaptionText 'Switch'; TextOff 'OFF'
      ProcessValue <- "GSV-511"
   TextField "Text field_4" at 277,170 size 75x23; Text 'GSV-511'
   Switch "Switch_3" at 361,216 size 64x32; TextOn 'ON'; CaptionText 'Switch'; TextOff 'OFF'
      ProcessValue <- "GSV-514"
   TextField "Text field_5" at 287,218 size 16x23; Text 'Text'
   TextField "Text field_6" at 281,218 size 75x23; Text 'GSV-514'
   Switch "Switch_4" at 361,264 size 64x32; TextOn 'ON'; CaptionText 'Switch'; TextOff 'OFF'
      ProcessValue <- "GSV-519"
   TextField "Text field_7" at 281,266 size 75x23; Text 'GSV-519'
   Switch "Switch_5" at 361,312 size 64x32; TextOn 'ON'; CaptionText 'Switch'; TextOff 'OFF'
      ProcessValue <- "GSV-521"
   TextField "Text field_8" at 281,314 size 75x23; Text 'GSV-521'
   Switch "Switch_6" at 529,163 size 64x32; TextOn 'ON'; CaptionText 'Switch'; TextOff 'OFF'
      ProcessValue <- "M001.ST"
   TextField "Text field_9" at 478,168 size 49x23; Text 'M001'
   Switch "Switch_7" at 536,296 size 64x32; TextOn 'ON'; CaptionText 'Switch'; TextOff 'OFF'
      ProcessValue <- "M003.ST"
   TextField "Text field_10" at 470,296 size 49x23; Text 'M003'
   Switch "Switch_8" at 536,221 size 64x32; TextOn 'ON'; CaptionText 'Switch'; TextOff 'OFF'
      ProcessValue <- "M002.ST"
   TextField "Text field_11" at 470,225 size 49x23; Text 'M002'
   IOField "I/O field_4" at 120,170 size 96x32; FormatPattern s999
      ProcessValue <- "TT-517"
   TextField "Text field_14" at 45,177 size 64x23; Text 'TT-517'
   IOField "I/O field_5" at 120,209 size 96x32; FormatPattern s999
      ProcessValue <- "TT-518"
   TextField "Text field_15" at 42,214 size 64x23; Text 'TT-518'
   Circle "Circle_1" at 623,154 size 48x48
      Visibility <- "M001.R"
   Circle "Circle_2" at 623,215 size 48x48
      Visibility <- "M002.R"
   Circle "Circle_3" at 623,276 size 48x48
      Visibility <- "M003.R"
   Bar "Bar_1" at 50,253 size 80x120; MinimumValue 0; MaximumValue 27648
      ProcessValue <- "LT-515"
   TextField "Text field_12" at 141,268 size 62x23; Text 'LT-515'
   IOField "I/O field_2" at 134,296 size 96x32; FormatPattern s999
      ProcessValue <- "LT-515"

screen "System screens" 800x480, template "Template_1"
   on GenerateScreen: SetTag("Tag_ScreenNumber", 2)
   Button "Back" at 1,52 size 159x47; TextOff 'Back'
      on Release: ActivateScreen("Root screen", 0)
   Button "HmiScreenItemData" at 36,146 size 159x47; TextOff 'SIMATIC PLC system diagnos...'; PictureOff "Navigates to SIMATIC PLC system diagnostics for KTP700 Basic+ PN 16.0.0.0"; PictureOn "Navigates to SIMATIC PLC system diagnostics for KTP700 Basic+ PN 16.0.0.0"
      on Release: ActivateScreen("SIMATIC PLC system diagnostics", 0)
   Button "HmiScreenItemData_1" at 36,205 size 159x47; TextOff 'Project information'; PictureOff "Navigates to Project information for KTP700 Basic+ PN 16.0.0.0"; PictureOn "Navigates to Project information for KTP700 Basic+ PN 16.0.0.0"
      on Release: ActivateScreen("Project information", 0)
   Button "HmiScreenItemData_2" at 36,264 size 159x47; TextOff 'User administration'; PictureOff "Navigates to User administration for KTP700 Basic+ PN 16.0.0.0"; PictureOn "Navigates to User administration for KTP700 Basic+ PN 16.0.0.0"
      on Release: ActivateScreen("User administration", 0)
   Button "HmiScreenItemData_3" at 36,323 size 159x47; TextOff 'System information'; PictureOff "Navigates to System information for KTP700 Basic+ PN 16.0.0.0"; PictureOn "Navigates to System information for KTP700 Basic+ PN 16.0.0.0"
      on Release: ActivateScreen("System information", 0)
   Button "HmiScreenItemData_4" at 207,146 size 159x47; TextOff 'Different jobs'; PictureOff "Navigates to Different jobs for KTP700 Basic+ PN 16.0.0.0"; PictureOn "Navigates to Different jobs for KTP700 Basic+ PN 16.0.0.0"
      on Release: ActivateScreen("Different jobs", 0)

screen "SIMATIC PLC system diagnostics" 800x480, template "Template_1"
   on GenerateScreen: SetTag("Tag_ScreenNumber", 3)
   SysDiagControl "HmiScreenItemData" at 1,100 size 796x321
   Button "Back" at 1,52 size 159x47; TextOff 'Back'
      on Release: ActivateScreen("System screens", 0)

screen "Project information" 800x480, template "Template_1"
   on GenerateScreen: SetTag("Tag_ScreenNumber", 4)
   TextField "HmiScreenItemData" at 35,102 size 171x28; Text 'Project name:'
   TextField "HmiScreenItemData_1" at 241,102 size 524x28; Text 'ChemicalProcess'
   TextField "HmiScreenItemData_2" at 35,132 size 171x28; Text 'Created on:'
   TextField "HmiScreenItemData_3" at 241,132 size 524x28; Text '5/25/2021 10:32:50 AM'
   TextField "HmiScreenItemData_4" at 35,162 size 171x28; Text 'Author:'
   TextField "HmiScreenItemData_5" at 241,162 size 524x28; Text 'mika3'
   TextField "HmiScreenItemData_6" at 35,192 size 171x28; Text 'Description:'
   TextField "HmiScreenItemData_7" at 241,192 size 524x28; Text '(not configured)'
   Button "Back" at 1,52 size 159x47; TextOff 'Back'
      on Release: ActivateScreen("System screens", 0)

screen "User administration" 800x480, template "Template_1"
   on GenerateScreen: SetTag("Tag_ScreenNumber", 5)
   UserView "HmiScreenItemData" at 1,100 size 796x321
   Button "Back" at 1,52 size 159x47; TextOff 'Back'
      on Release: ActivateScreen("System screens", 0)

screen "System information" 800x480, template "Template_1"
   on GenerateScreen: SetTag("Tag_ScreenNumber", 6)
   TextField "HmiScreenItemData" at 35,102 size 171x28; Text 'HMI device type:'
   TextField "HmiScreenItemData_1" at 241,102 size 524x28; Text 'KTP700 Basic+ PN 16.0.0.0'
   TextField "HmiScreenItemData_2" at 35,132 size 171x28; Text 'Connection:'
   TextField "HmiScreenItemData_3" at 241,132 size 524x28; Text 'PROFINET (X1)'
   TextField "HmiScreenItemData_4" at 35,162 size 171x28; Text 'PLC:'
   TextField "HmiScreenItemData_5" at 241,162 size 524x28; Text 'SIMATIC S7 1500'
   Button "Back" at 1,52 size 159x47; TextOff 'Back'
      on Release: ActivateScreen("System screens", 0)

screen "Different jobs" 800x480, template "Template_1"
   on GenerateScreen: SetTag("Tag_ScreenNumber", 7)
   Button "Online" at 36,146 size 159x47; TextOff 'Online'
      on Release: function_bb44b551(0)
   Button "Offline" at 36,205 size 159x47; TextOff 'Offline'
      on Release: function_bb44b551(1)
   Button "Transfer" at 36,264 size 159x47; TextOff 'Transfer'
      on Release: function_bb44b551(2)
   Button "Toggle language" at 36,323 size 159x47; TextOff 'Toggle language'
      on Release: function_fb9197e8(-1)
   Button "Stop Runtime" at 207,146 size 159x47; TextOff 'Stop Runtime'
      on Release: StopRuntime(0)
   Button "Back" at 1,52 size 159x47; TextOff 'Back'
      on Release: ActivateScreen("System screens", 0)
*)